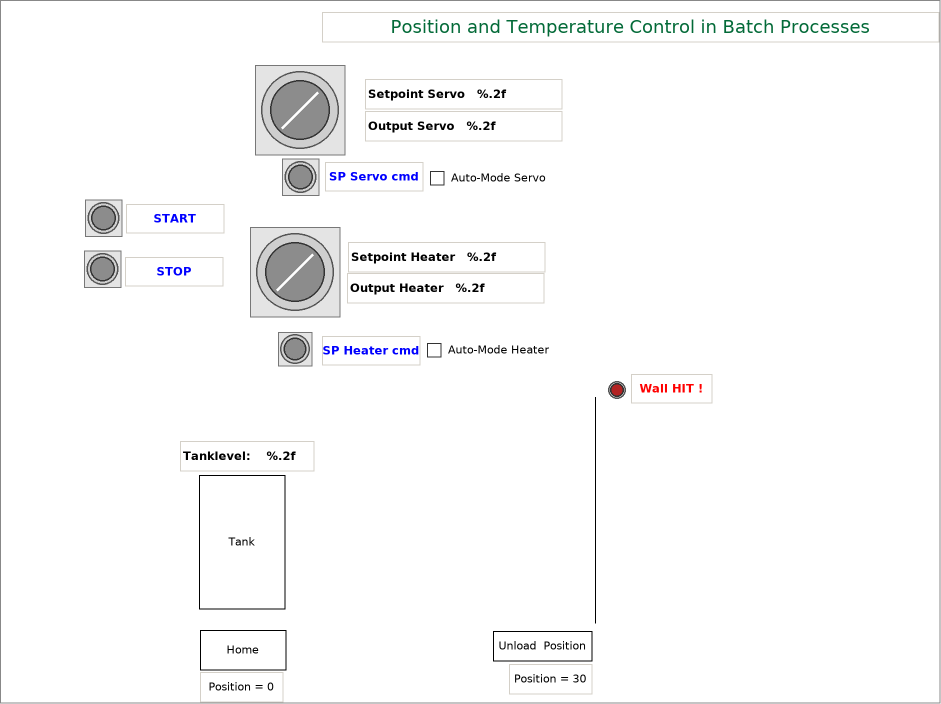
VISUALIZATION UserInterface  // 941x704
    PushSwitch (282,158 37x38), variable: GVL_IO.xPushButton1, behaviour: TAP, style: Switch-PushSwitch-Gray
    Potentiometer360 (255,65 90x90), variable: GVL_IO.SetPoint_ServoX, style: Potentiometer-Potentiometer360-Gray, scale format: %d, scale 0..60
        p2431819421: Outside
    Textfield (365,79 197x30), "Setpoint Servo %.2f", text variable: GVL_IO.SetPoint_ServoX
    Textfield (365,111 197x30), "Output Servo %.2f", text variable: GVL_IO.Output_ServoX
    Potentiometer360 (250,227 90x90), variable: GVL_IO.SetPointHeater, style: Potentiometer-Potentiometer360-Gray, scale format: %d, scale 0..100
        p2431819421: Outside
    PushSwitch (278,331 34x36), variable: GVL_IO.xPushButton2, behaviour: TAP, style: Switch-PushSwitch-Gray
    Textfield (348,242 197x30), "Setpoint Heater %.2f", text variable: GVL_IO.SetPointHeater
    Textfield (347,273 197x30), "Output Heater %.2f", text variable: GVL_IO.Output_Heater
    Rectangle (200,630 86x40), "Home"
    Rectangle (493,631 99x30), "Unload Position"
    Textfield (509,664 83x30), "Position = 30"
    Textfield (200,672 83x30), "Position = 0"
    Rectangle (199,475 86x134), "Tank"
        p3560616238: GVL_IO.Output_ServoX * 10
    Textfield (322,336 98x29), "SP Heater cmd"
    Textfield (325,162 98x29), "SP Servo cmd"
    Textfield (322,12 617x30), "Position and Temperature Control in Batch Processes"
    Textfield (180,441 134x30), "Tanklevel: %.2f", text variable: GVL_IO.TankLevelSensor
    Checkbox (425,340 125x20), "Auto-Mode Heater", variable: MAIN.PIDheater_on
    Checkbox (428,168 129x20), "Auto-Mode Servo", variable: MAIN.PIDServo_on
    Line (595,397) (595,623)
    Lamp1 (607,380 20x20), variable: (GVL_IO.Output_ServoX>31), style: Lamp-Lamp1-Red
    Textfield (631,374 81x29), "Wall HIT !", invisible if: (GVL_IO.Output_ServoX<=30.6)
    PushSwitch (85,199 37x38), variable: GVL_IO.StartPr, behaviour: TAP, style: Switch-PushSwitch-Gray
    PushSwitch (84,250 37x38), variable: GVL_IO.StopPr, behaviour: TAP, style: Switch-PushSwitch-Gray
    Textfield (126,204 98x29), "START"
    Textfield (125,257 98x29), "STOP"
END_VISUALIZATION

(* stored: Version 1.1.0.1, ProductVersion 3.1.4024.2
   Visu UserInterface: Id {8126f8ab-e6ef-48b6-9ba2-149e11247293} *)
